// TIA Portal V20 export
DATA_BLOCK "MotionNodes"   // DB39
// stored: Access Published, MemoryReserve 100, Namespace Unit1
   VAR
      MotionToPLC : "LER_typeMotionToPLC";
      PLCToMotion : "LER_typePLCToMotion";
   END_VAR
BEGIN
   PLCToMotion.Parameters.StackMain.Global.CPM := 30.0;
   PLCToMotion.Parameters.StackMain.Global.StageWidth := 240.0;
   PLCToMotion.Parameters.StackMain.Auto.CellCount := 39;
   PLCToMotion.Parameters.StackMain.Auto.InitialPosFinalRoller := 0.0;
   PLCToMotion.Parameters.StackMain.Auto.InitialPosCompensator := 0.0;
   PLCToMotion.Parameters.StackMain.Auto.InitialPosAnodePnPX1 := 0.0;
   PLCToMotion.Parameters.StackMain.Auto.InitialPosAnodePnPX2 := 0.0;
   PLCToMotion.Parameters.StackMain.Auto.InitialPosAnodePnPZ1 := 0.0;
   PLCToMotion.Parameters.StackMain.Auto.InitialPosAnodePnPZ2 := 0.0;
   PLCToMotion.Parameters.StackMain.Auto.InitialPosCathodePnPX1 := 0.0;
   PLCToMotion.Parameters.StackMain.Auto.InitialPosCathodePnPX2 := 0.0;
   PLCToMotion.Parameters.StackMain.Auto.InitialPosCathodePnPZ1 := 0.0;
   PLCToMotion.Parameters.StackMain.Auto.InitialPosCathodePnPZ2 := 0.0;
   PLCToMotion.Parameters.StackMain.Auto.InitialPosAnodeMandrelYFront := 50.0;
   PLCToMotion.Parameters.StackMain.Auto.InitialPosAnodeMandrelYRear := 50.0;
   PLCToMotion.Parameters.StackMain.Auto.InitialPosAnodeMandrelZFront := 50.0;
   PLCToMotion.Parameters.StackMain.Auto.InitialPosAnodeMandrelZRear := 50.0;
   PLCToMotion.Parameters.StackMain.Auto.InitialPosCathodeMandrelYFront := 50.0;
   PLCToMotion.Parameters.StackMain.Auto.InitialPosCathodeMandrelYRear := 50.0;
   PLCToMotion.Parameters.StackMain.Auto.InitialPosCathodeMandrelZFront := 50.0;
   PLCToMotion.Parameters.StackMain.Auto.InitialPosCathodeMandrelZRear := 50.0;
   PLCToMotion.Parameters.StackMain.Auto.Pos1FinalRollerXFwdOutputCam := 10.0;
   PLCToMotion.Parameters.StackMain.Auto.Pos1FinalRollerXBwdOutputCam := 10.0;
   PLCToMotion.Parameters.StackMain.Auto.Pos1FinalRollerXStackTableDownOutputCam := 140.0;
   PLCToMotion.Parameters.StackMain.Auto.Pos1FinalRollerXStackAnodeVisionOutputCam := 200.0;
   PLCToMotion.Parameters.StackMain.Auto.Pos1FinalRollerXStackCathodeVisionOutputCam := 300.0;
   PLCToMotion.Parameters.StackMain.Auto.Pos1AnodePnPX1FwdOutputCam := 10.0;
   PLCToMotion.Parameters.StackMain.Auto.Pos1AnodePnPX1BwdOutputCam := 10.0;
   PLCToMotion.Parameters.StackMain.Auto.Pos1AnodePnPX1ReelCutDataDeleteOffOutputCam := 10.0;
   PLCToMotion.Parameters.StackMain.Auto.Pos1AnodePnPX2FwdOutputCam := 10.0;
   PLCToMotion.Parameters.StackMain.Auto.Pos1AnodePnPX2BwdOutputCam := 10.0;
   PLCToMotion.Parameters.StackMain.Auto.Pos1AnodePnPZ1Down1OutputCam := 1.0;
   PLCToMotion.Parameters.StackMain.Auto.Pos1AnodePnPZ1Up1OutputCam := 1.0;
   PLCToMotion.Parameters.StackMain.Auto.Pos1AnodePnPZ2Down1OutputCam := 1.0;
   PLCToMotion.Parameters.StackMain.Auto.Pos1AnodePnPZ2Up1OutputCam := 1.0;
   PLCToMotion.Parameters.StackMain.Auto.Pos1AnodePnPZ1Down2OutputCam := 1.0;
   PLCToMotion.Parameters.StackMain.Auto.Pos1AnodePnPZ1Up2OutputCam := 1.0;
   PLCToMotion.Parameters.StackMain.Auto.Pos1AnodePnPZ2Down2OutputCam := 1.0;
   PLCToMotion.Parameters.StackMain.Auto.Pos1AnodePnPZ2Up2OutputCam := 1.0;
   PLCToMotion.Parameters.StackMain.Auto.Pos1AnodePnPZ1SuctionOnOutputCam := 15.0;
   PLCToMotion.Parameters.StackMain.Auto.Pos1AnodePnPZ1SuctionOffOutputCam := 25.0;
   PLCToMotion.Parameters.StackMain.Auto.Pos1AnodePnPZ1ReelCutBlowOutputCam := 15.0;
   PLCToMotion.Parameters.StackMain.Auto.Pos1AnodePnPZ1ReelCutDataDeleteOnOutputCam := 5.0;
   PLCToMotion.Parameters.StackMain.Auto.Pos1AnodePnPZ1AlignVisionOutputCam := 1.0;
   PLCToMotion.Parameters.StackMain.Auto.Pos1AnodePnPZ2SuctionOnOutputCam := 15.0;
   PLCToMotion.Parameters.StackMain.Auto.Pos1AnodePnPZ2SuctionOffOutputCam := 25.0;
   PLCToMotion.Parameters.StackMain.Auto.Pos1AnodeAlignSuctionOnOutputCam := 25.0;
   PLCToMotion.Parameters.StackMain.Auto.Pos1AnodeAlignSuctionOffOutputCam := 15.0;
   PLCToMotion.Parameters.StackMain.Auto.Pos1CathodePnPX1FwdOutputCam := 10.0;
   PLCToMotion.Parameters.StackMain.Auto.Pos1CathodePnPX1BwdOutputCam := 10.0;
   PLCToMotion.Parameters.StackMain.Auto.Pos1CathodePnPX1ReelCutDataDeleteOffOutputCam := 1.0;
   PLCToMotion.Parameters.StackMain.Auto.Pos1CathodePnPX2FwdOutputCam := 10.0;
   PLCToMotion.Parameters.StackMain.Auto.Pos1CathodePnPX2BwdOutputCam := 10.0;
   PLCToMotion.Parameters.StackMain.Auto.Pos1CathodePnPZ1Down1OutputCam := 1.0;
   PLCToMotion.Parameters.StackMain.Auto.Pos1CathodePnPZ1Up1OutputCam := 1.0;
   PLCToMotion.Parameters.StackMain.Auto.Pos1CathodePnPZ2Down1OutputCam := 1.0;
   PLCToMotion.Parameters.StackMain.Auto.Pos1CathodePnPZ2Up1OutputCam := 1.0;
   PLCToMotion.Parameters.StackMain.Auto.Pos1CathodePnPZ1Down2OutputCam := 1.0;
   PLCToMotion.Parameters.StackMain.Auto.Pos1CathodePnPZ1Up2OutputCam := 1.0;
   PLCToMotion.Parameters.StackMain.Auto.Pos1CathodePnPZ2Down2OutputCam := 1.0;
   PLCToMotion.Parameters.StackMain.Auto.Pos1CathodePnPZ2Up2OutputCam := 1.0;
   PLCToMotion.Parameters.StackMain.Auto.Pos1CathodePnPZ1SuctionOnOutputCam := 15.0;
   PLCToMotion.Parameters.StackMain.Auto.Pos1CathodePnPZ1SuctionOffOutputCam := 25.0;
   PLCToMotion.Parameters.StackMain.Auto.Pos1CathodePnPZ1ReelCutBlowOutputCam := 15.0;
   PLCToMotion.Parameters.StackMain.Auto.Pos1CathodePnPZ1ReelCutDataDeleteOnOutputCam := 5.0;
   PLCToMotion.Parameters.StackMain.Auto.Pos1CathodePnPZ1AlignVisionOutputCam := 1.0;
   PLCToMotion.Parameters.StackMain.Auto.Pos1CathodePnPZ2SuctionOnOutputCam := 15.0;
   PLCToMotion.Parameters.StackMain.Auto.Pos1CathodePnPZ2SuctionOffOutputCam := 25.0;
   PLCToMotion.Parameters.StackMain.Auto.Pos1CathodeAlignSuctionOnOutputCam := 25.0;
   PLCToMotion.Parameters.StackMain.Auto.Pos1CathodeAlignSuctionOffOutputCam := 15.0;
   PLCToMotion.Parameters.StackMain.Auto.Pos2FinalRollerXFwdOutputCam := 300.0;
   PLCToMotion.Parameters.StackMain.Auto.Pos2FinalRollerXBwdOutputCam := 300.0;
   PLCToMotion.Parameters.StackMain.Auto.Pos2FinalRollerXStackTableDownOutputCam := 200.0;
   PLCToMotion.Parameters.StackMain.Auto.Pos2FinalRollerXStackAnodeVisionOutputCam := 40.0;
   PLCToMotion.Parameters.StackMain.Auto.Pos2FinalRollerXStackCathodeVisionOutputCam := 330.0;
   PLCToMotion.Parameters.StackMain.Auto.Pos2AnodePnPX1FwdOutputCam := 530.0;
   PLCToMotion.Parameters.StackMain.Auto.Pos2AnodePnPX1BwdOutputCam := 530.0;
   PLCToMotion.Parameters.StackMain.Auto.Pos2AnodePnPX1ReelCutDataDeleteOffOutputCam := 530.0;
   PLCToMotion.Parameters.StackMain.Auto.Pos2AnodePnPX2FwdOutputCam := 530.0;
   PLCToMotion.Parameters.StackMain.Auto.Pos2AnodePnPX2BwdOutputCam := 530.0;
   PLCToMotion.Parameters.StackMain.Auto.Pos2AnodePnPZ1Down1OutputCam := 19.0;
   PLCToMotion.Parameters.StackMain.Auto.Pos2AnodePnPZ1Up1OutputCam := 19.0;
   PLCToMotion.Parameters.StackMain.Auto.Pos2AnodePnPZ2Down1OutputCam := 19.0;
   PLCToMotion.Parameters.StackMain.Auto.Pos2AnodePnPZ2Up1OutputCam := 19.0;
   PLCToMotion.Parameters.StackMain.Auto.Pos2AnodePnPZ1Down2OutputCam := 29.0;
   PLCToMotion.Parameters.StackMain.Auto.Pos2AnodePnPZ1Up2OutputCam := 29.0;
   PLCToMotion.Parameters.StackMain.Auto.Pos2AnodePnPZ2Down2OutputCam := 29.0;
   PLCToMotion.Parameters.StackMain.Auto.Pos2AnodePnPZ2Up2OutputCam := 29.0;
   PLCToMotion.Parameters.StackMain.Auto.Pos2AnodePnPZ1SuctionOnOutputCam := 20.0;
   PLCToMotion.Parameters.StackMain.Auto.Pos2AnodePnPZ1SuctionOffOutputCam := 30.0;
   PLCToMotion.Parameters.StackMain.Auto.Pos2AnodePnPZ1ReelCutBlowOutputCam := 20.0;
   PLCToMotion.Parameters.StackMain.Auto.Pos2AnodePnPZ1ReelCutDataDeleteOnOutputCam := 20.0;
   PLCToMotion.Parameters.StackMain.Auto.Pos2AnodePnPZ1AlignVisionOutputCam := 24.0;
   PLCToMotion.Parameters.StackMain.Auto.Pos2AnodePnPZ2SuctionOnOutputCam := 20.0;
   PLCToMotion.Parameters.StackMain.Auto.Pos2AnodePnPZ2SuctionOffOutputCam := 30.0;
   PLCToMotion.Parameters.StackMain.Auto.Pos2AnodeAlignSuctionOnOutputCam := 30.0;
   PLCToMotion.Parameters.StackMain.Auto.Pos2AnodeAlignSuctionOffOutputCam := 20.0;
   PLCToMotion.Parameters.StackMain.Auto.Pos2CathodePnPX1FwdOutputCam := 530.0;
   PLCToMotion.Parameters.StackMain.Auto.Pos2CathodePnPX1BwdOutputCam := 530.0;
   PLCToMotion.Parameters.StackMain.Auto.Pos2CathodePnPX1ReelCutDataDeleteOffOutputCam := 530.0;
   PLCToMotion.Parameters.StackMain.Auto.Pos2CathodePnPX2FwdOutputCam := 530.0;
   PLCToMotion.Parameters.StackMain.Auto.Pos2CathodePnPX2BwdOutputCam := 530.0;
   PLCToMotion.Parameters.StackMain.Auto.Pos2CathodePnPZ1Down1OutputCam := 19.0;
   PLCToMotion.Parameters.StackMain.Auto.Pos2CathodePnPZ1Up1OutputCam := 19.0;
   PLCToMotion.Parameters.StackMain.Auto.Pos2CathodePnPZ2Down1OutputCam := 19.0;
   PLCToMotion.Parameters.StackMain.Auto.Pos2CathodePnPZ2Up1OutputCam := 19.0;
   PLCToMotion.Parameters.StackMain.Auto.Pos2CathodePnPZ1Down2OutputCam := 29.0;
   PLCToMotion.Parameters.StackMain.Auto.Pos2CathodePnPZ1Up2OutputCam := 29.0;
   PLCToMotion.Parameters.StackMain.Auto.Pos2CathodePnPZ2Down2OutputCam := 29.0;
   PLCToMotion.Parameters.StackMain.Auto.Pos2CathodePnPZ2Up2OutputCam := 29.0;
   PLCToMotion.Parameters.StackMain.Auto.Pos2CathodePnPZ1SuctionOnOutputCam := 20.0;
   PLCToMotion.Parameters.StackMain.Auto.Pos2CathodePnPZ1SuctionOffOutputCam := 30.0;
   PLCToMotion.Parameters.StackMain.Auto.Pos2CathodePnPZ1ReelCutBlowOutputCam := 20.0;
   PLCToMotion.Parameters.StackMain.Auto.Pos2CathodePnPZ1ReelCutDataDeleteOnOutputCam := 20.0;
   PLCToMotion.Parameters.StackMain.Auto.Pos2CathodePnPZ1AlignVisionOutputCam := 24.0;
   PLCToMotion.Parameters.StackMain.Auto.Pos2CathodePnPZ2SuctionOnOutputCam := 20.0;
   PLCToMotion.Parameters.StackMain.Auto.Pos2CathodePnPZ2SuctionOffOutputCam := 30.0;
   PLCToMotion.Parameters.StackMain.Auto.Pos2CathodeAlignSuctionOnOutputCam := 30.0;
   PLCToMotion.Parameters.StackMain.Auto.Pos2CathodeAlignSuctionOffOutputCam := 20.0;
   PLCToMotion.Parameters.StackMain.StackCalculate.Position.FinalRollerBwdPos := 0.0;
   PLCToMotion.Parameters.StackMain.StackCalculate.Position.FinalRollerFwdPos := 75.0;
   PLCToMotion.TechnologyObject.OutputCam.FinalRollerXFwdOutputCam := 224;
   PLCToMotion.TechnologyObject.OutputCam.FinalRollerXBwdOutputCam := 225;
   PLCToMotion.TechnologyObject.OutputCam.FinalRollerXStackTableDownOutputCam := 206;
   PLCToMotion.TechnologyObject.OutputCam.FinalRollerXStackAnodeVisionOutputCam := 446;
   PLCToMotion.TechnologyObject.OutputCam.FinalRollerXStackCathodeVisionOutputCam := 445;
   PLCToMotion.TechnologyObject.OutputCam.AnodePnPX1FwdOutputCam := 413;
   PLCToMotion.TechnologyObject.OutputCam.AnodePnPX1BwdOutputCam := 412;
   PLCToMotion.TechnologyObject.OutputCam.AnodePnPX2FwdOutputCam := 415;
   PLCToMotion.TechnologyObject.OutputCam.AnodePnPX2BwdOutputCam := 414;
   PLCToMotion.TechnologyObject.OutputCam.AnodePnPZ1Down1OutputCam := 441;
   PLCToMotion.TechnologyObject.OutputCam.AnodePnPZ1Up1OutputCam := 420;
   PLCToMotion.TechnologyObject.OutputCam.AnodePnPZ2Down1OutputCam := 437;
   PLCToMotion.TechnologyObject.OutputCam.AnodePnPZ2Up1OutputCam := 438;
   PLCToMotion.TechnologyObject.OutputCam.AnodePnPZ1Down2OutputCam := 430;
   PLCToMotion.TechnologyObject.OutputCam.AnodePnPZ1Up2OutputCam := 432;
   PLCToMotion.TechnologyObject.OutputCam.AnodePnPZ2Down2OutputCam := 436;
   PLCToMotion.TechnologyObject.OutputCam.AnodePnPZ2Up2OutputCam := 434;
   PLCToMotion.TechnologyObject.OutputCam.AnodePnPZ1SuctionOnOutputCam := 433;
   PLCToMotion.TechnologyObject.OutputCam.AnodePnPZ1SuctionOffOutputCam := 431;
   PLCToMotion.TechnologyObject.OutputCam.AnodePnPZ1ReelCutBlowOutputCam := 185;
   PLCToMotion.TechnologyObject.OutputCam.AnodePnPZ2SuctionOnOutputCam := 435;
   PLCToMotion.TechnologyObject.OutputCam.AnodePnPZ2SuctionOffOutputCam := 442;
   PLCToMotion.TechnologyObject.OutputCam.AnodeAlignSuctionOnOutputCam := 455;
   PLCToMotion.TechnologyObject.OutputCam.AnodeAlignSuctionOffOutputCam := 456;
   PLCToMotion.TechnologyObject.OutputCam.AnodePnPZ1ReelCutDataDeleteOnOutputCam := 134;
   PLCToMotion.TechnologyObject.OutputCam.AnodePnP1XReelCutDataDeleteOffOutputCam := 140;
   PLCToMotion.TechnologyObject.OutputCam.AnodeAlignVisionOutputCam := 187;
   PLCToMotion.TechnologyObject.OutputCam.CathodePnPX1FwdOutputCam := 417;
   PLCToMotion.TechnologyObject.OutputCam.CathodePnPX1BwdOutputCam := 416;
   PLCToMotion.TechnologyObject.OutputCam.CathodePnPX2FwdOutputCam := 418;
   PLCToMotion.TechnologyObject.OutputCam.CathodePnPX2BwdOutputCam := 419;
   PLCToMotion.TechnologyObject.OutputCam.CathodePnPZ1Down1OutputCam := 422;
   PLCToMotion.TechnologyObject.OutputCam.CathodePnPZ1Up1OutputCam := 423;
   PLCToMotion.TechnologyObject.OutputCam.CathodePnPZ2Down1OutputCam := 428;
   PLCToMotion.TechnologyObject.OutputCam.CathodePnPZ2Up1OutputCam := 429;
   PLCToMotion.TechnologyObject.OutputCam.CathodePnPZ1Down2OutputCam := 421;
   PLCToMotion.TechnologyObject.OutputCam.CathodePnPZ1Up2OutputCam := 439;
   PLCToMotion.TechnologyObject.OutputCam.CathodePnPZ2Down2OutputCam := 427;
   PLCToMotion.TechnologyObject.OutputCam.CathodePnPZ2Up2OutputCam := 425;
   PLCToMotion.TechnologyObject.OutputCam.CathodePnPZ1SuctionOnOutputCam := 457;
   PLCToMotion.TechnologyObject.OutputCam.CathodePnPZ1SuctionOffOutputCam := 443;
   PLCToMotion.TechnologyObject.OutputCam.CathodePnPZ1ReelCutBlowOutputCam := 424;
   PLCToMotion.TechnologyObject.OutputCam.CathodePnPZ2SuctionOnOutputCam := 426;
   PLCToMotion.TechnologyObject.OutputCam.CathodePnPZ2SuctionOffOutputCam := 444;
   PLCToMotion.TechnologyObject.OutputCam.CathodeAlignSuctionOnOutputCam := 440;
   PLCToMotion.TechnologyObject.OutputCam.CathodeAlignSuctionOffOutputCam := 458;
   PLCToMotion.TechnologyObject.OutputCam.CathodePnPZ1ReelCutDataDeleteOnOutputCam := 182;
   PLCToMotion.TechnologyObject.OutputCam.CathodePnP1XReelCutDataDeleteOffOutputCam := 186;
   PLCToMotion.TechnologyObject.OutputCam.CathodeAlignVisionOutputCam := 195;
END_DATA_BLOCK
